    movej(get_inverse_kin(pose_trans(Pallet_prepick_p, get_tcp_offset()), qnear=Pallet_prepick_q), a=1.3962634015954636, v=1.0471975511965976)
    $ 851 "MoveL"
    $ 852 "Pick_canister" "breakAfter"
    movel(pose_trans(Pick_canister_p, get_tcp_offset()), a=1.2, v=0.25)
    $ 853 "Set OuTNET_Gripper=6"
    write_output_integer_register(0, 6)
    $ 854 "Set OutNet_Tool=On"
    write_output_boolean_register(2, True)
    $ 855 "Wait: 3.0"
    sleep(3.0)
    $ 856 "Wait InNET_InPos=HI"
    while (read_input_boolean_register(1) == False):
      sync()
    end
    $ 857 "Set OutNet_Tool=Off"
    write_output_boolean_register(2, False)
    $ 858 "MoveL"
    $ 859 "Pallet_prepick" "breakAfter"
    movel(pose_trans(Pallet_prepick_p, get_tcp_offset()), a=1.2, v=0.25)
    $ 860 "MoveJ"
    $ 861 "Canister_aprox" "breakAfter"
    movej(get_inverse_kin(Canister_aprox_p, qnear=Canister_aprox_q), a=1.3962634015954636, v=1.0471975511965976)
    $ 862 "MoveL"
    $ 863 "pl1Canister34up" "breakAfter"
    movel(pose_trans(Plane_1_Pack, pose_trans(p[.061451264231, -.289311417922, -.073379282729, -.000157706105, .000169116670, 2.356123162082], pl1Canister34up_p)), a=1.2, v=0.25)
    $ 864 "MoveL"
    $ 865 "pl1Canister34" "breakAfter"
    movel(pose_trans(Plane_1_Pack, pose_trans(p[.061451264231, -.289311417922, -.073379282729, -.000157706105, .000169116670, 2.356123162082], pl1Canister34_p)), a=1.2, v=0.25)
    $ 866 "Set OuTNET_Gripper=2"
    write_output_integer_register(0, 2)
    $ 867 "Set OutNet_Tool=On"
    write_output_boolean_register(2, True)
    $ 868 "Wait: 3.0"
    sleep(3.0)
    $ 869 "Wait InNET_InPos=HI"
    while (read_input_boolean_register(1) == False):
      sync()
    end
    $ 870 "Set OutNet_Tool=Off"
    write_output_boolean_register(2, False)
    $ 871 "MoveL"
    $ 872 "pl1Canist34up" "breakAfter"
    movel(pose_trans(Plane_1_Pack, pose_trans(p[.061451264231, -.289311417922, -.073379282729, -.000157706105, .000169116670, 2.356123162082], pl1Canist34up_p)), a=1.2, v=0.25)
    $ 873 "MoveJ"
    $ 874 "Canister_aprox" "breakAfter"
    movej(get_inverse_kin(Canister_aprox_p, qnear=Canister_aprox_q), a=1.3962634015954636, v=1.0471975511965976)
  end
  def Plane1_Packs():
    $ 875 "Plane1_Packs" "noBreak"
    $ 876 "MoveJ"
    $ 877 "PL1orig" "breakAfter"
    movej(get_inverse_kin(PL1orig_p, qnear=PL1orig_q), a=1.3962634015954636, v=1.0471975511965976, r=0.05)
    $ 878 "PL1_Xinc" "breakAfter"
    movej(get_inverse_kin(PL1_Xinc_p, qnear=PL1_Xinc_q), a=1.3962634015954636, v=1.0471975511965976)
    $ 879 "PL1_Yinc" "breakAfter"
    movej(get_inverse_kin(PL1_Yinc_p, qnear=PL1_Yinc_q), a=1.3962634015954636, v=1.0471975511965976)
    $ 880 "PL1orig_aprox" "breakAfter"
    movej(get_inverse_kin(PL1orig_aprox_p, qnear=PL1orig_aprox_q), a=1.3962634015954636, v=1.0471975511965976)
  end
  def Plane2_Charger():
    $ 881 "Plane2_Charger" "noBreak"
    $ 882 "MoveJ"
    $ 883 "PL2orig" "breakAfter"
    movej(get_inverse_kin(PL2orig_p, qnear=PL2orig_q), a=1.3962634015954636, v=1.0471975511965976)
    $ 884 "PL2orig_aprox" "breakAfter"
    movej(get_inverse_kin(PL2orig_aprox_p, qnear=PL2orig_aprox_q), a=1.3962634015954636, v=1.0471975511965976)
    $ 885 "PL2_Xinc" "breakAfter"
    movej(get_inverse_kin(PL2_Xinc_p, qnear=PL2_Xinc_q), a=1.3962634015954636, v=1.0471975511965976)
    $ 886 "PL2_Yinc" "breakAfter"
    movej(get_inverse_kin(PL2_Yinc_p, qnear=PL2_Yinc_q), a=1.3962634015954636, v=1.0471975511965976)
  end
  def Plane3_C1move():
    $ 887 "Plane3_C1move" "noBreak"
    $ 888 "MoveJ"
    $ 889 "PL3orig" "breakAfter"
    movej(get_inverse_kin(PL3orig_p, qnear=PL3orig_q), a=1.3962634015954636, v=1.0471975511965976)
    $ 890 "PL3orig_aprox" "breakAfter"
    movej(get_inverse_kin(PL3orig_aprox_p, qnear=PL3orig_aprox_q), a=1.3962634015954636, v=1.0471975511965976)
    $ 891 "PL3_Yinc" "breakAfter"
    movej(get_inverse_kin(PL3_Yinc_p, qnear=PL3_Yinc_q), a=1.3962634015954636, v=1.0471975511965976)
    $ 892 "PL3_Zinc" "breakAfter"
    movej(get_inverse_kin(PL3_Zinc_p, qnear=PL3_Zinc_q), a=1.3962634015954636, v=1.0471975511965976)
  end
  def Plane4_C2move():
    $ 893 "Plane4_C2move" "noBreak"
    $ 894 "MoveJ"
    $ 895 "PL4orig" "breakAfter"
    movej(get_inverse_kin(PL4orig_p, qnear=PL4orig_q), a=1.3962634015954636, v=1.0471975511965976)
    $ 896 "PL4_Yinc" "breakAfter"
    movej(get_inverse_kin(PL4_Yinc_p, qnear=PL4_Yinc_q), a=1.3962634015954636, v=1.0471975511965976)
    $ 897 "PL4_Zinc" "breakAfter"
    movej(get_inverse_kin(PL4_Zinc_p, qnear=PL4_Zinc_q), a=1.3962634015954636, v=1.0471975511965976)
    $ 898 "pl4orig_aprox" "breakAfter"
    movej(get_inverse_kin(pl4orig_aprox_p, qnear=pl4orig_aprox_q), a=1.3962634015954636, v=1.0471975511965976)
  end
  def mm_cam_check():
    $ 899 "mm_cam_check" "noBreak"
    $ 900 "Switch mm_bay"
    switch_1 = mm_bay
    $ 901 "Case 1"
    if (1 == switch_1):
      $ 902 "MoveL"
      $ 903 "Waypoint_4" "breakAfter"
      movel(Waypoint_4_p, a=1.2, v=0.25)
      $ 904 "MoveJ"
      $ 905 "Waypoint_1" "breakAfter"
      movej(get_inverse_kin(Waypoint_1_p, qnear=Waypoint_1_q), a=1.3962634015954636, v=1.0471975511965976)
      $ 906 "Wait: 2.0"
      sleep(2.0)
      $ 907 "Set mm_pht_rdy_stp=1"
      modbus_set_output_register("mm_pht_rdy_stp", 1)
      $ 908 "Wait mm_pht_stp_done≥1 and mm_pht_stp_done≤1"
      while (not(modbus_get_signal_status("mm_pht_stp_done") >= 1  and  modbus_get_signal_status("mm_pht_stp_done") <= 1)):
        sync()
      end
      $ 909 "Waypoint_6" "breakAfter"
      movel(Waypoint_6_p, a=1.2, v=0.25)
      $ 910 "Waypoint_8" "breakAfter"
      movel(Waypoint_8_p, a=1.2, v=0.25)
      $ 911 "Wait: 2.0"
      sleep(2.0)
      $ 912 "Set mm_pht_rdy_stp=2"
      modbus_set_output_register("mm_pht_rdy_stp", 2)
      $ 913 "Wait mm_pht_stp_done≤2 and mm_pht_stp_done≥2"
      while (not(modbus_get_signal_status("mm_pht_stp_done") <= 2  and  modbus_get_signal_status("mm_pht_stp_done") >= 2)):
        sync()
      end
      $ 914 "Set mm_pht_rdy_stp=0"
      modbus_set_output_register("mm_pht_rdy_stp", 0)
      $ 915 "Wait: 2.0"
      sleep(2.0)
    end
  end
  def mm_p1_put_back():
    $ 916 "mm_p1_put_back" "noBreak"
    $ 917 "MoveJ"
    $ 918 "Pack_aprox_1" "breakAfter"
    movej(get_inverse_kin(Pack_aprox_1_p, qnear=Pack_aprox_1_q), a=1.3962634015954636, v=1.0471975511965976)
    $ 919 "MoveL"
    $ 920 "Waypoint_3" "breakAfter"
    movel(Waypoint_3_p, a=1.2, v=0.25)
    $ 921 "Set OuTNET_Gripper=0"
    write_output_integer_register(0, 0)
    $ 922 "Set OutNet_Tool=On"
    write_output_boolean_register(2, True)
    $ 923 "Wait: 2.0"
    sleep(2.0)
    $ 924 "Waypoint_2" "breakAfter"
    movel(Waypoint_2_p, a=1.2, v=0.25)
    $ 925 "Set OutNet_Tool=Off"
    write_output_boolean_register(2, False)
    $ 926 "'put back done, fix containers next'"
    # 'put back done, fix containers next'
  end
  def mm_get_poke():
    $ 927 "mm_get_poke" "noBreak"
    $ 928 "MoveJ"
    $ 929 "UL_Pack_aprox_1" "breakAfter"
    movej(get_inverse_kin(UL_Pack_aprox_1_p, qnear=UL_Pack_aprox_1_q), a=1.3962634015954636, v=1.0471975511965976)
    $ 930 "abv_poke" "breakAfter"
    movej(get_inverse_kin(abv_poke_p, qnear=abv_poke_q), a=1.3962634015954636, v=1.0471975511965976)
    $ 931 "Set OuTNET_Gripper=2"
    write_output_integer_register(0, 2)
    $ 932 "Set OutNet_Tool=On"
    write_output_boolean_register(2, True)
    $ 933 "Wait: 2.0"
    sleep(2.0)
    $ 934 "Wait InNET_InPos=HI"
    while (read_input_boolean_register(1) == False):
      sync()
    end
    $ 935 "Set OutNet_Tool=Off"
    write_output_boolean_register(2, False)
    $ 936 "'open gripper'"
    # 'open gripper'
    $ 937 "poke_holder" "breakAfter"
    movej(get_inverse_kin(poke_holder_p, qnear=poke_holder_q), a=1.3962634015954636, v=1.0471975511965976)
    $ 938 "Set OuTNET_Gripper=6"
    write_output_integer_register(0, 6)
    $ 939 "Set OutNet_Tool=On"
    write_output_boolean_register(2, True)
    $ 940 "Wait: 3.5"
    sleep(3.5)
    $ 941 "Wait InNET_InPos=HI"
    while (read_input_boolean_register(1) == False):
      sync()
    end
    $ 942 "Set OutNet_Tool=Off"
    write_output_boolean_register(2, False)
    $ 943 "'close_gripper'"
    # 'close_gripper'
    $ 944 "abv_poke" "breakAfter"
    movej(get_inverse_kin(abv_poke_p, qnear=abv_poke_q), a=1.3962634015954636, v=1.0471975511965976)
    $ 945 "UL_Pack_aprox_1" "breakAfter"
    movej(get_inverse_kin(UL_Pack_aprox_1_p, qnear=UL_Pack_aprox_1_q), a=1.3962634015954636, v=1.0471975511965976)
  end
  def mm_fix_pack1():
    $ 946 "mm_fix_pack1" "noBreak"
    $ 947 "MoveJ"
    $ 948 "UL_Pack_aprox_1" "breakAfter"
    movej(get_inverse_kin(UL_Pack_aprox_1_p, qnear=UL_Pack_aprox_1_q), a=1.3962634015954636, v=1.0471975511965976)
    $ 949 "abv_p1" "breakAfter"
    movej(get_inverse_kin(abv_p1_p, qnear=abv_p1_q), a=1.3962634015954636, v=1.0471975511965976)
    $ 950 "MoveL"
    $ 951 "If c1_recorrect≟1"
    if (modbus_get_signal_status("c1_recorrect") == 1):
      $ 952 "c1_approx" "breakAfter"
      movel(c1_approx_p, a=1.2, v=0.25)
      $ 953 "c1_push" "breakAfter"
      movel(c1_push_p, a=1.2, v=0.25)
      $ 954 "c1_approx" "breakAfter"
      movel(c1_approx_p, a=1.2, v=0.25)
      $ 955 "'Fixed c1'"
      # 'Fixed c1'
      $ 956 "abv_p1" "breakAfter"
      movel(abv_p1_p, a=1.2, v=0.25)
    end
    $ 957 "If c2_recorrect≟1"
    if (modbus_get_signal_status("c2_recorrect") == 1):
      $ 958 "c2_approx" "breakAfter"
      movel(c2_approx_p, a=1.2, v=0.25)
      $ 959 "c2_push" "breakAfter"
      movel(c2_push_p, a=1.2, v=0.25)
      $ 960 "c2_approx" "breakAfter"
      movel(c2_approx_p, a=1.2, v=0.25)
      $ 961 "'Fixed c2'"
      # 'Fixed c2'
      $ 962 "abv_p1" "breakAfter"
      movel(abv_p1_p, a=1.2, v=0.25)
    end
    $ 963 "If c3_reconnect≟1"
    if (modbus_get_signal_status("c3_reconnect") == 1):
      $ 964 "c3_approx" "breakAfter"
      movel(c3_approx_p, a=1.2, v=0.25)
      $ 965 "c3_push" "breakAfter"
      movel(c3_push_p, a=1.2, v=0.25)
      $ 966 "c3_approx" "breakAfter"
      movel(c3_approx_p, a=1.2, v=0.25)
      $ 967 "'Fixed c3'"
      # 'Fixed c3'
      $ 968 "abv_p1" "breakAfter"
      movel(abv_p1_p, a=1.2, v=0.25)
    end
    $ 969 "If c4_reconnect≟1"
    if (modbus_get_signal_status("c4_reconnect") == 1):
      $ 970 "c4_approx" "breakAfter"
      movel(c4_approx_p, a=1.2, v=0.25)
      $ 971 "c4_push" "breakAfter"
      movel(c4_push_p, a=1.2, v=0.25)
      $ 972 "c4_approx" "breakAfter"
      movel(c4_approx_p, a=1.2, v=0.25)
      $ 973 "'Fixed c4'"
      # 'Fixed c4'
      $ 974 "abv_p1" "breakAfter"
      movel(abv_p1_p, a=1.2, v=0.25)
    end
  end
  def mm_drop_poke():
    $ 975 "mm_drop_poke" "noBreak"
    $ 976 "MoveJ"
    $ 977 "UL_Pack_aprox_1" "breakAfter"
    movej(get_inverse_kin(UL_Pack_aprox_1_p, qnear=UL_Pack_aprox_1_q), a=1.3962634015954636, v=1.0471975511965976)
    $ 978 "abv_poke" "breakAfter"
    movej(get_inverse_kin(abv_poke_p, qnear=abv_poke_q), a=1.3962634015954636, v=1.0471975511965976)
    $ 979 "poke_holder" "breakAfter"
    movej(get_inverse_kin(poke_holder_p, qnear=poke_holder_q), a=1.3962634015954636, v=1.0471975511965976)
    $ 980 "Set OuTNET_Gripper=2"
    write_output_integer_register(0, 2)
    $ 981 "Set OutNet_Tool=On"
    write_output_boolean_register(2, True)
    $ 982 "Wait InNET_InPos=HI"
    while (read_input_boolean_register(1) == False):
      sync()
    end
    $ 983 "Set OutNet_Tool=Off"
    write_output_boolean_register(2, False)
    $ 984 "abv_poke" "breakAfter"
    movej(get_inverse_kin(abv_poke_p, qnear=abv_poke_q), a=1.3962634015954636, v=1.0471975511965976)
    $ 985 "Set OuTNET_Gripper=0"
    write_output_integer_register(0, 0)
    $ 986 "Set OutNet_Tool=On"
    write_output_boolean_register(2, True)
    $ 987 "Waypoint_5" "breakAfter"
    movej(get_inverse_kin(Waypoint_5_p, qnear=Waypoint_5_q), a=1.3962634015954636, v=1.0471975511965976)
    $ 988 "Set OutNet_Tool=Off"
    write_output_boolean_register(2, False)
  end
  $ 2 "BeforeStart"
  $ 3 "CurrentPos≔get_actual_tcp_pose()"
  global CurrentPos= get_actual_tcp_pose ()
  $ 4 "CurrentXValue≔CurrentPos[0]"
  global CurrentXValue=CurrentPos[0]
  $ 5 "CurrentYValue≔CurrentPos[1]"
  global CurrentYValue=CurrentPos[1]
  $ 6 "CurrentZValue≔CurrentPos[2]"
  global CurrentZValue=CurrentPos[2]
  $ 7 "mm_bay≔0"
  global mm_bay=0
  $ 8 "m_innet_op≔2000"
  global m_innet_op=2000
  $ 9 "Popup: Press Continue. If modbus error occurs go to Installation > Fieldbus > Modbus > 'refresh list' before proceeding. Check Raspberry pi is on. Using SSH, run 'sudo pm2 start 0 && sudo pm2 logs 0' if errors persist. This prompt is not an error but a warning."
  popup("Press Continue. If modbus error occurs go to Installation > Fieldbus > Modbus > 'refresh list' before proceeding. Check Raspberry pi is on. Using SSH, run 'sudo pm2 start 0 && sudo pm2 logs 0' if errors persist. This prompt is not an error but a warning.", "Message", False, False, blocking=True)
  $ 10 "mm_lst_insp_id≔mm_insp_id"
  global mm_lst_insp_id=modbus_get_signal_status("mm_insp_id")
  $ 11 "mm_lst_res_v≔mm_res_ver"
  global mm_lst_res_v=modbus_get_signal_status("mm_res_ver")
  $ 12 "mm_lat_c1r≔ False "
  global mm_lat_c1r=  False
  $ 13 "mm_lat_c2r≔ False "
  global mm_lat_c2r=  False
  $ 14 "mm_lat_c3r≔ False "
  global mm_lat_c3r=  False
  $ 15 "mm_lat_c4r≔ False "
  global mm_lat_c4r=  False
  $ 16 "mm_recorr_req≔ False "
  global mm_recorr_req=  False
  $ 17 "Set mm_pht_rdy_stp=0"
  modbus_set_output_register("mm_pht_rdy_stp", 0)
  $ 18 "Set mm_recv_inst=0"
  modbus_set_output_register("mm_recv_inst", 0)
  $ 19 "If (CurrentXValue≥-0.018 and CurrentXValue ≤-0.014) and (CurrentYValue≤-0.296 and CurrentYValue≥-0.310) and (CurrentZValue≥0.160 and CurrentZValue≤0.305)"
  if ((CurrentXValue >= -0.018  and  CurrentXValue  <= -0.014)  and  (CurrentYValue <= -0.296  and  CurrentYValue >= -0.310)  and  (CurrentZValue >= 0.160  and  CurrentZValue <= 0.305)):
    $ 20 "Popup: Robot inside warehouse, press continue to bring it to a safe position automatically."
    popup("Robot inside warehouse, press continue to bring it to a safe position automatically.", "Message", False, False, blocking=True)
    $ 21 "CurrentPos[0]=-0.106"
    CurrentPos[0]=-0.106
    $ 22 "CurrentPos[1]=-0.211"
    CurrentPos[1]=-0.211
    $ 23 "MoveL"
    $ 24 "CurrentPos" "breakAfter"
    movel(CurrentPos, a=1.2, v=0.25)
    $ 25 "MoveJ"
    $ 26 "ChargerSafe" "breakAfter"
    movej(get_inverse_kin(ChargerSafe_p, qnear=ChargerSafe_q), a=1.3962634015954636, v=1.0471975511965976)
    $ 27 "UL_HomePos" "breakAfter"
    movej(get_inverse_kin(UL_HomePos_p, qnear=UL_HomePos_q), a=1.3962634015954636, v=1.0471975511965976)
  end
  while (True):
    $ 28 "Robot Program"
    $ 29 "mm_bay≔0"
    global mm_bay=0
    $ 30 "Set mm_pht_rdy_stp=0"
    modbus_set_output_register("mm_pht_rdy_stp", 0)
    $ 31 "Set mm_recv_inst=0"
    modbus_set_output_register("mm_recv_inst", 0)
    $ 32 "Set OutNET_Done=Off"
    write_output_boolean_register(1, False)
    $ 33 "Set OutNet_FullBin=Off"
    write_output_boolean_register(3, False)
    $ 34 "Set OutNet_Tool=Off"
    write_output_boolean_register(2, False)
    $ 35 "Set OuTNET_Gripper=0"
    write_output_integer_register(0, 0)
    $ 36 "Set OutNET_Ready=On"
    write_output_boolean_register(0, True)
    $ 37 "Wait: 1.0"
    sleep(1.0)
    $ 38 "Set mm_done=Off"
    write_output_boolean_register(31, False)
    $ 39 "MoveJ"
    $ 40 "UL_HomePos" "breakAfter"
    movej(get_inverse_kin(UL_HomePos_p, qnear=UL_HomePos_q), a=1.3962634015954636, v=1.0471975511965976)
    $ 41 "Loop"
    while (True):
      $ 42 "Set OutNET_Done=Off"
      write_output_boolean_register(1, False)
      $ 43 "Wait: 0.5"
      sleep(0.5)
      $ 44 "Wait InNET_Enable"
      while (not(read_input_boolean_register(2))):
        sync()
      end
      $ 45 "Wait InNET_Run and InNET_Operation≠0"
      while (not(read_input_boolean_register(0)  and  read_input_integer_register(0) != 0)):
        sync()
      end
      $ 46 "m_innet_op≔InNET_Operation"
      global m_innet_op=read_input_integer_register(0)
      $ 47 "Switch InNET_Operation"
      switch_1 = read_input_integer_register(0)
      $ 48 "Case 1"
      if (1 == switch_1):
        $ 49 "Wait InNET_Enable and InNet_Halt"
        while (not(read_input_boolean_register(2)  and  read_input_boolean_register(3))):
          sync()
        end
        $ 50 "Set OutNET_Done=Off"
        write_output_boolean_register(1, False)
        $ 51 "Call CHARGER1_pick"
        CHARGER1_pick()
        $ 52 "Set OutNET_Done=On"
        write_output_boolean_register(1, True)
        $ 53 "Wait: 2.0"
        sleep(2.0)
      elif (2 == switch_1):
        $ 54 "Case 2"
        $ 55 "Wait InNET_Enable and  InNet_Halt"
        while (not(read_input_boolean_register(2)  and   read_input_boolean_register(3))):
          sync()
        end
        $ 56 "Set OutNET_Done=Off"
        write_output_boolean_register(1, False)
        $ 57 "Call C1pk2move"
        C1pk2move()
        $ 58 "Call CHARGER1_pick"
        CHARGER1_pick()
        $ 59 "Set OutNET_Done=On"
        write_output_boolean_register(1, True)
        $ 60 "Wait: 2.0"
        sleep(2.0)
      elif (3 == switch_1):
        $ 61 "Case 3"
        $ 62 "Wait InNET_Enable and InNet_Halt"
        while (not(read_input_boolean_register(2)  and  read_input_boolean_register(3))):
          sync()
        end
        $ 63 "Set OutNET_Done=Off"
        write_output_boolean_register(1, False)
        $ 64 "Call C1pk3move"
        C1pk3move()
        $ 65 "Call CHARGER1_pick"
        CHARGER1_pick()
        $ 66 "Set OutNET_Done=On"
        write_output_boolean_register(1, True)
        $ 67 "Wait: 2.0"
        sleep(2.0)
      elif (4 == switch_1):
        $ 68 "Case 4"
        $ 69 "Wait InNET_Enable and InNet_Halt"
        while (not(read_input_boolean_register(2)  and  read_input_boolean_register(3))):
          sync()
        end
        $ 70 "Set OutNET_Done=Off"
        write_output_boolean_register(1, False)
        $ 71 "Call C1pk4move"
        C1pk4move()
        $ 72 "Call CHARGER1_pick"
        CHARGER1_pick()
        $ 73 "Set OutNET_Done=On"
        write_output_boolean_register(1, True)
        $ 74 "Wait: 2.0"
        sleep(2.0)
      elif (5 == switch_1):
        $ 75 "Case 5"
        $ 76 "Wait InNET_Enable and InNet_Halt"
        while (not(read_input_boolean_register(2)  and  read_input_boolean_register(3))):
          sync()
        end
        $ 77 "Set OutNET_Done=Off"
        write_output_boolean_register(1, False)
        $ 78 "Call C1pk5move"
        C1pk5move()
        $ 79 "Call CHARGER1_pick"
        CHARGER1_pick()
        $ 80 "Set OutNET_Done=On"
        write_output_boolean_register(1, True)
        $ 81 "Wait: 2.0"
        sleep(2.0)
      elif (6 == switch_1):
        $ 82 "Case 6"
        $ 83 "Wait InNET_Enable and InNet_Halt"
        while (not(read_input_boolean_register(2)  and  read_input_boolean_register(3))):
          sync()
        end
        $ 84 "Set OutNET_Done=Off"
        write_output_boolean_register(1, False)
        $ 85 "Call PACK1_release"
        PACK1_release()
        $ 86 "Set OutNET_Done=On"
        write_output_boolean_register(1, True)
        $ 87 "Wait: 2.0"
        sleep(2.0)
      elif (7 == switch_1):
        $ 88 "Case 7"
        $ 89 "Wait InNET_Enable and InNet_Halt"
        while (not(read_input_boolean_register(2)  and  read_input_boolean_register(3))):
          sync()
        end
        $ 90 "Set OutNET_Done=Off"
        write_output_boolean_register(1, False)
        $ 91 "Call PACK2_release"
        PACK2_release()
        $ 92 "Set OutNET_Done=On"
        write_output_boolean_register(1, True)
        $ 93 "Wait: 2.0"
        sleep(2.0)
      elif (8 == switch_1):
        $ 94 "Case 8"
        $ 95 "Wait InNET_Enable and InNet_Halt"
        while (not(read_input_boolean_register(2)  and  read_input_boolean_register(3))):
          sync()
        end
        $ 96 "Set OutNET_Done=Off"
        write_output_boolean_register(1, False)
        $ 97 "Call PACK3_release"
        PACK3_release()
        $ 98 "Set OutNET_Done=On"
        write_output_boolean_register(1, True)
        $ 99 "Wait: 2.0"
        sleep(2.0)
      elif (9 == switch_1):
        $ 100 "Case 9"
        $ 101 "Wait InNET_Enable and InNet_Halt"
        while (not(read_input_boolean_register(2)  and  read_input_boolean_register(3))):
          sync()
        end
        $ 102 "Set OutNET_Done=Off"
        write_output_boolean_register(1, False)
        $ 103 "Call PK1CAN1_release"
        PK1CAN1_release()
        $ 104 "Call PALLET__remove"
        PALLET__remove()
        $ 105 "Set OutNET_Done=On"
        write_output_boolean_register(1, True)
        $ 106 "Wait: 2.0"
        sleep(2.0)
      elif (10 == switch_1):
        $ 107 "Case 10"
        $ 108 "Wait InNET_Enable and InNet_Halt"
        while (not(read_input_boolean_register(2)  and  read_input_boolean_register(3))):
          sync()
        end
        $ 109 "Set OutNET_Done=Off"
        write_output_boolean_register(1, False)
        $ 110 "Call PK1CAN2_release"
        PK1CAN2_release()
        $ 111 "Call PALLET__remove"
        PALLET__remove()
        $ 112 "Set OutNET_Done=On"
        write_output_boolean_register(1, True)
        $ 113 "Wait: 2.0"
        sleep(2.0)
      elif (11 == switch_1):
        $ 114 "Case 11"
        $ 115 "Wait InNET_Enable and InNet_Halt"
        while (not(read_input_boolean_register(2)  and  read_input_boolean_register(3))):
          sync()
        end
        $ 116 "Set OutNET_Done=Off"
        write_output_boolean_register(1, False)
        $ 117 "Call PK1CAN3_release"
        PK1CAN3_release()
        $ 118 "Call PALLET__remove"
        PALLET__remove()
        $ 119 "Set OutNET_Done=On"
        write_output_boolean_register(1, True)
        $ 120 "Wait: 2.0"
        sleep(2.0)
      elif (12 == switch_1):
        $ 121 "Case 12"
        $ 122 "Wait InNET_Enable and InNet_Halt"
        while (not(read_input_boolean_register(2)  and  read_input_boolean_register(3))):
          sync()
        end
        $ 123 "Set OutNET_Done=Off"
        write_output_boolean_register(1, False)
        $ 124 "Call PK1CAN4_release"
        PK1CAN4_release()
        $ 125 "Call PALLET__remove"
        PALLET__remove()
        $ 126 "Set OutNET_Done=On"
        write_output_boolean_register(1, True)
        $ 127 "Wait: 2.0"
        sleep(2.0)
      elif (13 == switch_1):
        $ 128 "Case 13"
        $ 129 "Wait InNET_Enable and InNet_Halt"
        while (not(read_input_boolean_register(2)  and  read_input_boolean_register(3))):
          sync()
        end
        $ 130 "Set OutNET_Done=Off"
        write_output_boolean_register(1, False)
        $ 131 "Call PK2CAN1_release"
        PK2CAN1_release()
        $ 132 "Call PALLET__remove"
        PALLET__remove()
        $ 133 "Set OutNET_Done=On"
        write_output_boolean_register(1, True)
        $ 134 "Wait: 2.0"
        sleep(2.0)
      elif (14 == switch_1):
        $ 135 "Case 14"
        $ 136 "Wait InNET_Enable and InNet_Halt"
        while (not(read_input_boolean_register(2)  and  read_input_boolean_register(3))):
          sync()
        end
        $ 137 "Set OutNET_Done=Off"
        write_output_boolean_register(1, False)
        $ 138 "Call PK2CAN2_release"
        PK2CAN2_release()
        $ 139 "Call PALLET__remove"
        PALLET__remove()
        $ 140 "Set OutNET_Done=On"
        write_output_boolean_register(1, True)
        $ 141 "Wait: 2.0"
        sleep(2.0)
      elif (15 == switch_1):
        $ 142 "Case 15"
        $ 143 "Wait InNET_Enable and InNet_Halt"
        while (not(read_input_boolean_register(2)  and  read_input_boolean_register(3))):
          sync()
        end
        $ 144 "Set OutNET_Done=Off"
        write_output_boolean_register(1, False)
        $ 145 "Call PK2CAN3_release"
        PK2CAN3_release()
        $ 146 "Call PALLET__remove"
        PALLET__remove()
        $ 147 "Set OutNET_Done=On"
        write_output_boolean_register(1, True)
        $ 148 "Wait: 2.0"
        sleep(2.0)
      elif (16 == switch_1):
        $ 149 "Case 16"
        $ 150 "Wait InNET_Enable and InNet_Halt"
        while (not(read_input_boolean_register(2)  and  read_input_boolean_register(3))):
          sync()
        end
        $ 151 "Set OutNET_Done=Off"
        write_output_boolean_register(1, False)
        $ 152 "Call PK2CAN4_release"
        PK2CAN4_release()
        $ 153 "Call PALLET__remove"
        PALLET__remove()
        $ 154 "Set OutNET_Done=On"
        write_output_boolean_register(1, True)
        $ 155 "Wait: 2.0"
        sleep(2.0)
      elif (17 == switch_1):
        $ 156 "Case 17"
        $ 157 "Wait InNET_Enable"
        while (not(read_input_boolean_register(2))):
          sync()
        end
        $ 158 "Set OutNET_Done=Off"
        write_output_boolean_register(1, False)
        $ 159 "Call PK3CAN1_release"
        PK3CAN1_release()
        $ 160 "Call PALLET__remove"
        PALLET__remove()
        $ 161 "Set OutNET_Done=On"
        write_output_boolean_register(1, True)
        $ 162 "Wait: 2.0"
        sleep(2.0)
      elif (18 == switch_1):
        $ 163 "Case 18"
        $ 164 "Wait InNET_Enable and InNet_Halt"
        while (not(read_input_boolean_register(2)  and  read_input_boolean_register(3))):
          sync()
        end
        $ 165 "Set OutNET_Done=Off"
        write_output_boolean_register(1, False)
        $ 166 "Call PK3CAN2_release"
        PK3CAN2_release()
        $ 167 "Call PALLET__remove"
        PALLET__remove()
        $ 168 "Set OutNET_Done=On"
        write_output_boolean_register(1, True)
        $ 169 "Wait: 2.0"
        sleep(2.0)
      elif (19 == switch_1):
        $ 170 "Case 19"
        $ 171 "Wait InNET_Enable and InNet_Halt"
        while (not(read_input_boolean_register(2)  and  read_input_boolean_register(3))):
          sync()
        end
        $ 172 "Set OutNET_Done=Off"
        write_output_boolean_register(1, False)
        $ 173 "Call PK3CAN3_release"
        PK3CAN3_release()
        $ 174 "Call PALLET__remove"
        PALLET__remove()
        $ 175 "Set OutNET_Done=On"
        write_output_boolean_register(1, True)
        $ 176 "Wait: 2.0"
        sleep(2.0)
      elif (20 == switch_1):
        $ 177 "Case 20"
        $ 178 "Wait InNET_Enable and InNet_Halt"
        while (not(read_input_boolean_register(2)  and  read_input_boolean_register(3))):
          sync()
        end
        $ 179 "Set OutNET_Done=Off"
        write_output_boolean_register(1, False)
        $ 180 "Call PK3CAN4_release"
        PK3CAN4_release()
        $ 181 "Call PALLET__remove"
        PALLET__remove()
        $ 182 "Set OutNET_Done=On"
        write_output_boolean_register(1, True)
        $ 183 "Wait: 2.0"
        sleep(2.0)
      elif (21 == switch_1):
        $ 184 "Case 21"
        $ 185 "Wait InNET_Enable and InNet_Halt"
        while (not(read_input_boolean_register(2)  and  read_input_boolean_register(3))):
          sync()
        end
        $ 186 "Set OutNET_Done=Off"
        write_output_boolean_register(1, False)
        $ 187 "Set OutNET_Done=On"
        write_output_boolean_register(1, True)
        $ 188 "Set OutNet_Tool=Off"
        write_output_boolean_register(2, False)
        $ 189 "Set mm_done=Off"
        write_output_boolean_register(31, False)
        $ 190 "mm_bay≔1"
        global mm_bay=1
        $ 191 "Call PACK1_pick"
        PACK1_pick()
        $ 192 "Set mm_recv_inst=1"
        modbus_set_output_register("mm_recv_inst", 1)
        $ 193 "Wait: 0.5"
        sleep(0.5)
        $ 194 "Set mm_recv_inst=0"
        modbus_set_output_register("mm_recv_inst", 0)
        $ 195 "Call mm_cam_check"
        mm_cam_check()
        $ 196 "If c1_recorrect≟ True  or c2_recorrect≟ True  or c3_reconnect≟ True  or c4_reconnect≟ True "
        if (modbus_get_signal_status("c1_recorrect") ==   True    or  modbus_get_signal_status("c2_recorrect") ==   True    or  modbus_get_signal_status("c3_reconnect") ==   True    or  modbus_get_signal_status("c4_reconnect") ==   True  ):
          $ 197 "Call mm_p1_put_back"
          mm_p1_put_back()
          $ 198 "Call mm_get_poke"
          mm_get_poke()
          $ 199 "Call mm_fix_pack1"
          mm_fix_pack1()
          $ 200 "Call mm_drop_poke"
          mm_drop_poke()
          $ 201 "Call PACK1_pick"
          PACK1_pick()
        end
        $ 202 "Call PACK_Unload"
        PACK_Unload()
        $ 203 "Set OutNET_Done=On"
        write_output_boolean_register(1, True)
        $ 204 "Wait: 2.0"
        sleep(2.0)
      elif (22 == switch_1):
        $ 205 "Case 22"
        $ 206 "Wait InNET_Enable and InNet_Halt"
        while (not(read_input_boolean_register(2)  and  read_input_boolean_register(3))):
          sync()
        end
        $ 207 "Set OutNET_Done=Off"
        write_output_boolean_register(1, False)
        $ 208 "Set OutNET_Done=On"
        write_output_boolean_register(1, True)
        $ 209 "mm_bay≔2"
        global mm_bay=2
        $ 210 "Call PACK2_pick"
        PACK2_pick()
        $ 211 "Call PACK_Unload"
        PACK_Unload()
        $ 212 "Set OutNET_Done=On"
        write_output_boolean_register(1, True)
        $ 213 "Wait: 2.0"
        sleep(2.0)
      elif (23 == switch_1):
        $ 214 "Case 23"
        $ 215 "Wait InNET_Enable and InNet_Halt"
        while (not(read_input_boolean_register(2)  and  read_input_boolean_register(3))):
          sync()
        end
        $ 216 "Set OutNET_Done=Off"
        write_output_boolean_register(1, False)
        $ 217 "Set OutNET_Done=On"
        write_output_boolean_register(1, True)
        $ 218 "mm_bay≔3"
        global mm_bay=3
        $ 219 "Call PACK3_pick"
        PACK3_pick()
        $ 220 "Call PACK_Unload"
        PACK_Unload()
        $ 221 "Set OutNET_Done=On"
        write_output_boolean_register(1, True)
        $ 222 "Wait: 2.0"
        sleep(2.0)
      end
    end
  end
end
